PROGRAM POUNCPowerOn
VAR
	fbXAxisPowerOn : MC_Power;
	fbXAxisDrive : MC_MoveRelative;
	DegreesToRelativeMovment_0: DegreesToRelativeMovment;
	HomingActive: BOOL;
	MC_Home_0: MC_Home;
	StartHoming: BOOL;
	endSW: BOOL;
	MC_Reset_0: MC_Reset;
	reset: BOOL;
	
	
	//command : STRING;
END_VAR

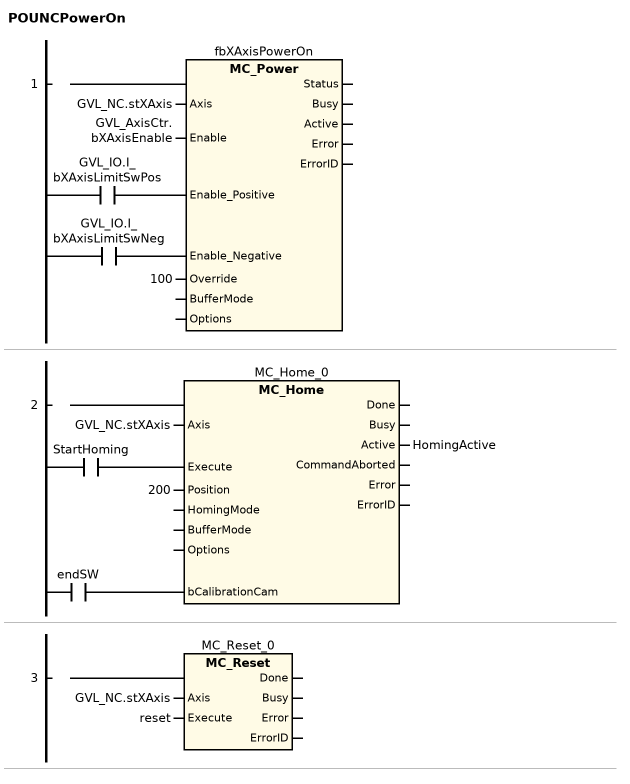
// NETWORK 1
fbXAxisPowerOn(
    Axis := GVL_NC.stXAxis,
    Enable := GVL_AxisCtr.bXAxisEnable,
    Enable_Positive := GVL_IO.I_bXAxisLimitSwPos,
    Enable_Negative := GVL_IO.I_bXAxisLimitSwNeg,
    Override := 100); // MC_Power

// NETWORK 2
MC_Home_0(
    Axis := GVL_NC.stXAxis,
    Execute := StartHoming,
    Position := 200,
    bCalibrationCam := endSW,
    Active => HomingActive); // MC_Home

// NETWORK 3
MC_Reset_0(Axis := GVL_NC.stXAxis, Execute := reset); // MC_Reset

END_PROGRAM

(* stored: Version 1.1.0.1, ProductVersion 3.1.4024.3
   POU POUNCPowerOn: Id {518f66f2-a21f-4a9a-84b8-3594f5178ae2}, SpecialFunc None *)
